(* Schneider Machine Expert - Basic project m4 to m5-9, file version 2.0.0.0 *)
(* ProjectInformations: Name=New project *)

HARDWARE
  Cpu 0: TM221CE16R
  EthernetConfiguration: NetworkName=M221, IpAllocationMode=FixedAddress, IpAddress=0.0.0.0, SubnetMask=0.0.0.0
  SerialLineConfiguration: Baud=Baud19200, Parity=ParityEven, DataBits=DataBits8, StopBits=StopBits1, PhysicalMedium=PhysicalMediumRs485, TransmissionMode=TransmissionModeModbusRtu, SlaveId=1, Addressing=SlaveAddressing
  MastTask: UsePeriodScanMode=false, PeriodScan=100
  FastTask: Period=255
  CpuBehavior: StartingMode=StartAsPreviousState, AutoSaveRamOnEeprom=true, WatchdogPeriod=250

SYMBOLS  (address, symbol, comment, settings)

POU New POU
  (* SectionNumber=0 *)

// Rung 0
  LD %M4
  ST %M2
  // as ST:
  //   %M2 := %M4;

// Rung 1
  LD %M4
  ST %M6
  // as ST:
  //   %M6 := %M4;

// Rung 2
  LD %M4
  ST %M7
  // as ST:
  //   %M7 := %M4;

// Rung 3
  LD %M4
  ST %M8
  // as ST:
  //   %M8 := %M4;

// Rung 4
  LD %M4
  ST %M9
  // as ST:
  //   %M9 := %M4;
